{attribute 'qualified_only'}
{attribute 'strict'}
TYPE EWPMaterial :
(
	black := 1,
	white := 2,
	metallic :=3,
	undetermined :=4,
	enum_member := 0
);
END_TYPE

(* stored: Version 1.1.0.1, ProductVersion 3.1.4024.9
   DUT EWPMaterial: Id {7ebc950e-59ce-4e5a-9ac0-3d460b1ba642} *)
